TYPE E_Mode :
(
	eMode_Initial,
	eMode_Secure,
	eMode_Reset,
	eMode_Stop,
	eMode_Manual,
	eMode_SemiAutomatic,
	eMode_FullyAutomatic
);
END_TYPE

(* stored: Version 1.1.0.1
   DUT E_Mode: Id {e98a56f5-c551-4329-9551-8ffa87381e28} *)
